// Mitsubishi GX Works2 project: Project34   PLC: FX3G

// global labels: Global1
VAR_GLOBAL
  StartA AT X010 : BOOL;
  SEN_IN AT X001 : BOOL;
  SEN_OUT AT X004 : BOOL;
  SEN_30 AT X003 : BOOL;
  SEN_15 AT X002 : BOOL;
  help1 AT M1 : BOOL;
END_VAR
VAR_GLOBAL CONSTANT
  Time1 : INT := 10;
  Time2 : INT := 10;
END_VAR
VAR_GLOBAL
  yuval AT X006 : BOOL;
END_VAR
VAR_GLOBAL CONSTANT
  Time3 : INT := 40;
END_VAR
VAR_GLOBAL
  ZILUF2 AT TS3 : BOOL;
  HELP3 AT M2 : BOOL;
  StartCoating AT X006 : BOOL;
  analogInput1 AT D8280 : INT;
  saveAnalogInput1 AT D8201 : INT;
END_VAR
VAR_GLOBAL CONSTANT
  topBound1 : INT := 5;
  topBound2 : INT := 10;
  lowerBound2 : INT := 6;
  Time4 : INT := 50;
END_VAR
VAR_GLOBAL
  CoatingLamp AT Y003 : BOOL;
  kkk1 AT Y002 : BOOL;
  kkk7 AT Y002 : BOOL;
  GFDKDN AT Y005 : BOOL;
  StartPacking AT X000 : BOOL;
  CreamStock AT D1100 : INT;
  UpdateCream AT D1200 : INT;
END_VAR
VAR_GLOBAL CONSTANT
  MinCream : INT := 300;
END_VAR
VAR_GLOBAL
  ChocolateStock AT D2100 : INT;
END_VAR
VAR_GLOBAL CONSTANT
  MinChocolate : INT := 240;
END_VAR
VAR_GLOBAL
  BiscuitStock AT D3100 : INT;
  UpdateBiscuit AT D3200 : INT;
END_VAR
VAR_GLOBAL CONSTANT
  MinBiscuit : INT := 6;
END_VAR
VAR_GLOBAL
  StartProcess AT X007 : BOOL;
  Check AT Y007 : BOOL;
  Coil5 AT M5 : BOOL;
  TransferCream AT X011 : BOOL;
  SprinklingContainer AT D4100 : INT;
  UpdateSprinkling AT D4200 : INT;
  ImmersionContainer AT D5100 : INT;
END_VAR
VAR_GLOBAL CONSTANT
  CreamUsed : INT := 300;
  NormalCoating : INT := 120;
  DoubleCoating : INT := 240;
  Init : INT;
  Unit : INT := 400;
END_VAR
VAR_GLOBAL
  Input AT D6000 : INT;
  UpdateChocolate AT D2300 : INT;
  UpdateImmersion AT D5300 : INT;
  BDIKA AT M8 : BOOL;
  DANUS AT M9 : BOOL;
  pack AT X000 : BOOL;
  Counter1 AT CC1 : BOOL;
END_VAR
VAR_GLOBAL CONSTANT
  counterVal1 : INT := 5;
END_VAR
VAR_GLOBAL
  Counter2 AT CC2 : BOOL;
END_VAR
VAR_GLOBAL CONSTANT
  counterVal2 : INT := 6;
END_VAR
VAR_GLOBAL
  Counter2output AT CS2 : BOOL;
  packCoil AT Y002 : BOOL;
  Krembows AT D3333 : INT;
END_VAR
VAR_GLOBAL CONSTANT
  addKrembow : INT := 6;
  Tens : INT := 10;
END_VAR
VAR_GLOBAL
  Coil12 AT M12 : BOOL;
  Coil13 AT M13 : BOOL;
END_VAR
VAR_GLOBAL CONSTANT
  Time5 : INT := 30;
END_VAR
VAR_GLOBAL
  Timer5 AT TC5 : BOOL;
  Coil14 AT M14 : BOOL;
  Coil15 AT M15 : BOOL;
  Timer6 AT TC6 : BOOL;
END_VAR
VAR_GLOBAL CONSTANT
  Time6 : INT := 10;
END_VAR
VAR_GLOBAL
  Timer7 AT TC7 : BOOL;
  Timer7Output AT TS7 : BOOL;
  Coil16 AT M16 : BOOL;
  Coil17 AT M17 : BOOL;
  Coil18 AT M18 : BOOL;
  Coil19 AT M19 : BOOL;
  Coil20 AT M20 : BOOL;
  Coil21 AT M21 : BOOL;
  Coil22 AT M22 : BOOL;
END_VAR
VAR_GLOBAL CONSTANT
  BiscuitUsed : INT := 6;
END_VAR
VAR_GLOBAL
  AnalogOutput AT D8282 : INT;
  Counter_Update AT CC8 : BOOL;
  Counter_Update6 AT CC9 : BOOL;
  Coil23 AT M23 : BOOL;
  Coil24 AT M24 : BOOL;
  Coil25 AT M25 : BOOL;
  Coil26 AT M26 : BOOL;
  WorkingDay AT Y007 : BOOL;
  Timer5Output AT TS5 : BOOL;
  Timer6Output AT TS6 : BOOL;
  DozensKrembows AT D4444 : INT;
  SprinklerFault AT X005 : BOOL;
  SprinklingLamp AT Y004 : BOOL;
  Timer3 AT TC3 : BOOL;
  Timer3Output AT TS3 : BOOL;
  Timer1 AT TC1 : BOOL;
  Timer1Output AT TS1 : BOOL;
  Timer2 AT TC2 : BOOL;
  Timer2Output AT TS2 : BOOL;
  ShinuaLamp1 AT Y000 : BOOL;
  ShinuaLamp2 AT Y001 : BOOL;
  Coil10 AT M10 : BOOL;
  Coil11 AT M11 : BOOL;
  Timer4 AT TC4 : BOOL;
  Timer4Output AT TS4 : BOOL;
  Counter1output AT CS1 : BOOL;
  Coil0 AT M0 : BOOL;
  coil27 AT M27 : BOOL;
END_VAR
VAR_GLOBAL CONSTANT
  Multiplier : INT := 40;
END_VAR
VAR_GLOBAL
  Coil28 AT M28 : BOOL;
END_VAR

// task Task_01 (event TRUE, interval 0, priority 31): POU_01

PROGRAM POU_01
(* structured ladder/FBD written out as ST: instructions are called as NAME(EN, inputs, outputs); _pN, _eN, _tN stand for wires *)
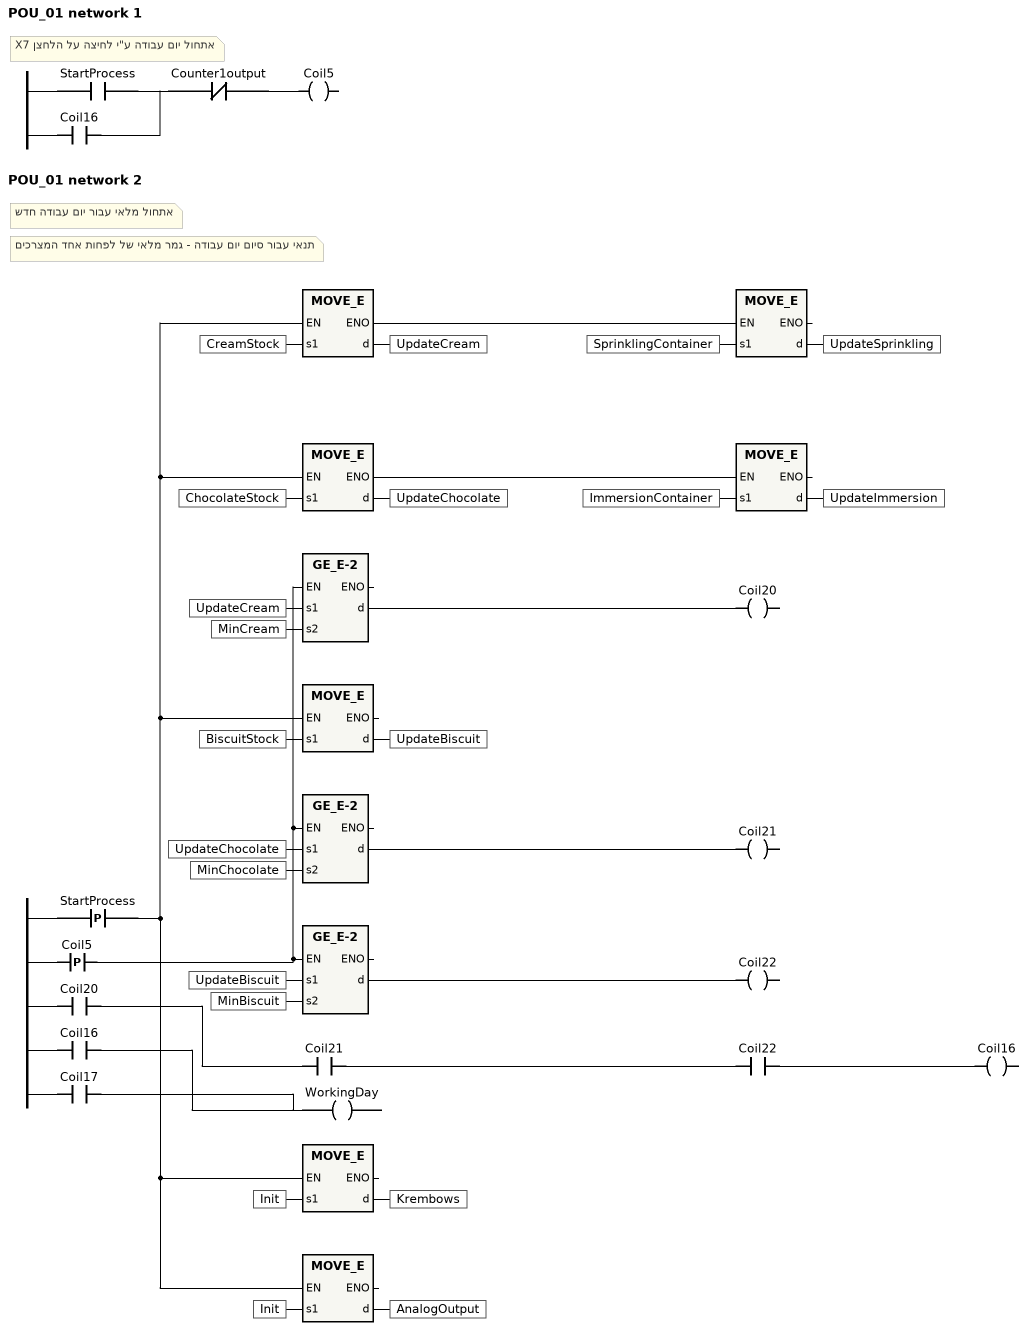
(* network 1 *)
(* אתחול יום עבודה ע"י לחיצה על הלחצן X7 *)
Coil5 := (StartProcess OR Coil16) AND NOT Counter1output;
(* network 2 *)
(* אתחול מלאי עבור יום עבודה חדש *)
(* תנאי עבור סיום יום עבודה - גמר מלאי של לפחות אחד המצרכים *)
_p1 := LDP(TRUE, StartProcess);
_e2 := MOVE_E(_p1, CreamStock, UpdateCream);
MOVE_E(_e2, SprinklingContainer, UpdateSprinkling);
_e3 := MOVE_E(_p1, ChocolateStock, UpdateChocolate);
MOVE_E(_e3, ImmersionContainer, UpdateImmersion);
MOVE_E(_p1, BiscuitStock, UpdateBiscuit);
MOVE_E(_p1, Init, Krembows);
MOVE_E(_p1, Init, AnalogOutput);
_p4 := LDP(TRUE, Coil5);
GE_E(_p4, UpdateCream, MinCream, _t5);
Coil20 := _t5;
GE_E(_p4, UpdateChocolate, MinChocolate, _t6);
Coil21 := _t6;
GE_E(_p4, UpdateBiscuit, MinBiscuit, _t7);
Coil22 := _t7;
Coil16 := Coil20 AND Coil21 AND Coil22;
WorkingDay := Coil16 OR Coil17;
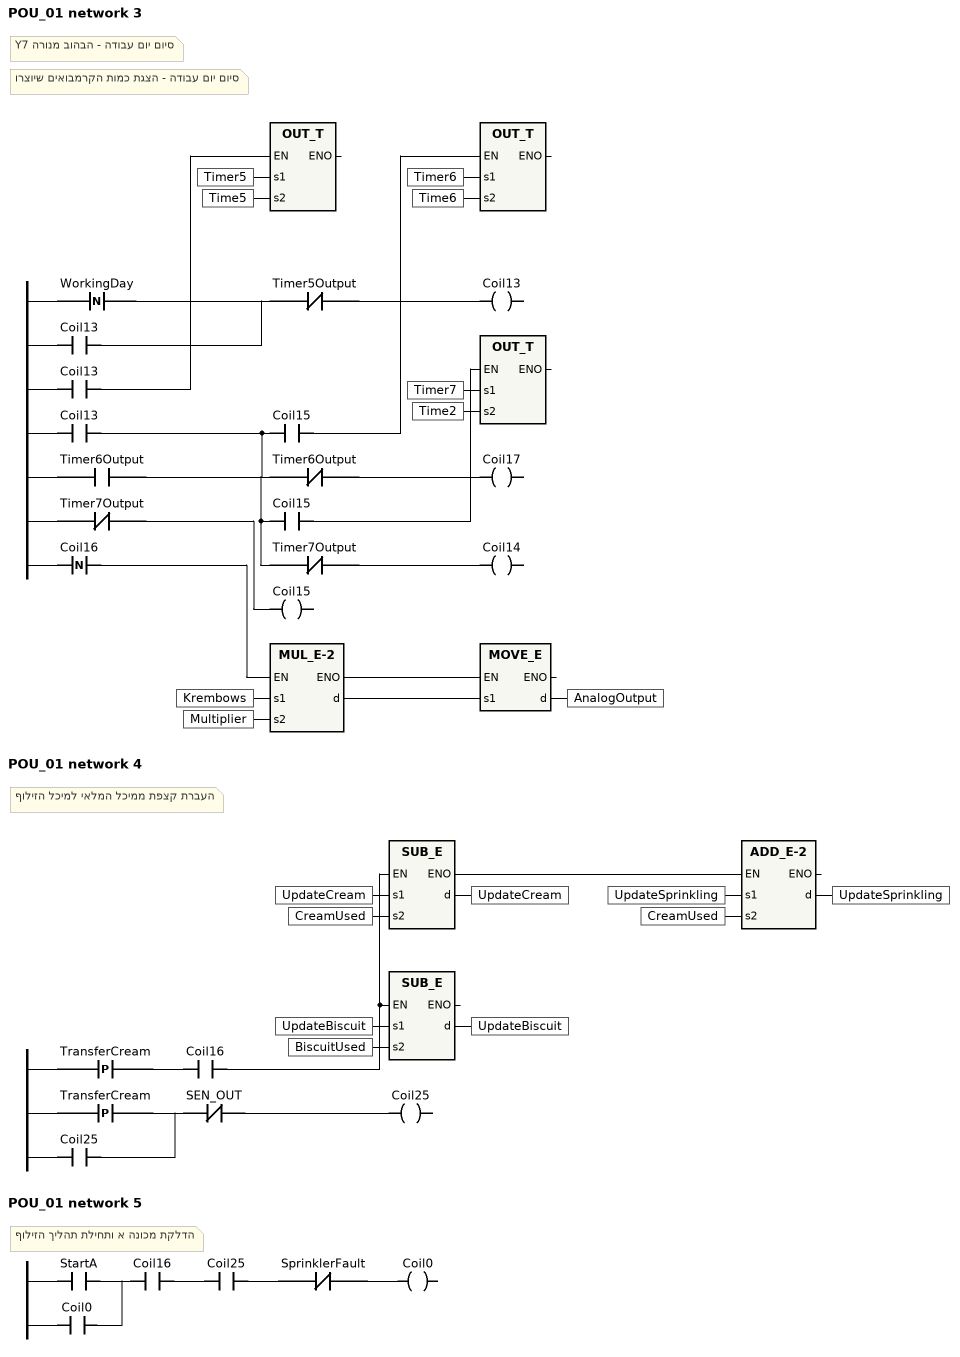
(* network 3 *)
(* סיום יום עבודה - הבהוב מנורה Y7 *)
(* סיום יום עבודה - הצגת כמות הקרמבואים שיוצרו *)
Coil13 := (LDF(TRUE, WorkingDay) OR Coil13) AND NOT Timer5Output;
OUT_T(Coil13, Timer5, Time5);
OUT_T(Coil13 AND Coil15, Timer6, Time6);
Coil17 := Coil13 AND NOT Timer6Output;
OUT_T(Timer6Output AND Coil15, Timer7, Time2);
Coil14 := Timer6Output AND NOT Timer7Output;
Coil15 := NOT Timer7Output;
_e2 := MUL_E(LDF(TRUE, Coil16), Krembows, Multiplier, _t1);
MOVE_E(_e2, _t1, AnalogOutput);
(* network 4 *)
(* העברת קצפת ממיכל המלאי למיכל הזילוף *)
_p1 := LDP(TRUE, TransferCream) AND Coil16;
_e2 := SUB_E(_p1, UpdateCream, CreamUsed, UpdateCream);
ADD_E(_e2, UpdateSprinkling, CreamUsed, UpdateSprinkling);
SUB_E(_p1, UpdateBiscuit, BiscuitUsed, UpdateBiscuit);
Coil25 := (LDP(TRUE, TransferCream) OR Coil25) AND NOT SEN_OUT;
(* network 5 *)
(* הדלקת מכונה א ותחילת תהליך הזילוף *)
Coil0 := (((StartA OR Coil0) AND Coil16) AND Coil25) AND NOT SprinklerFault;
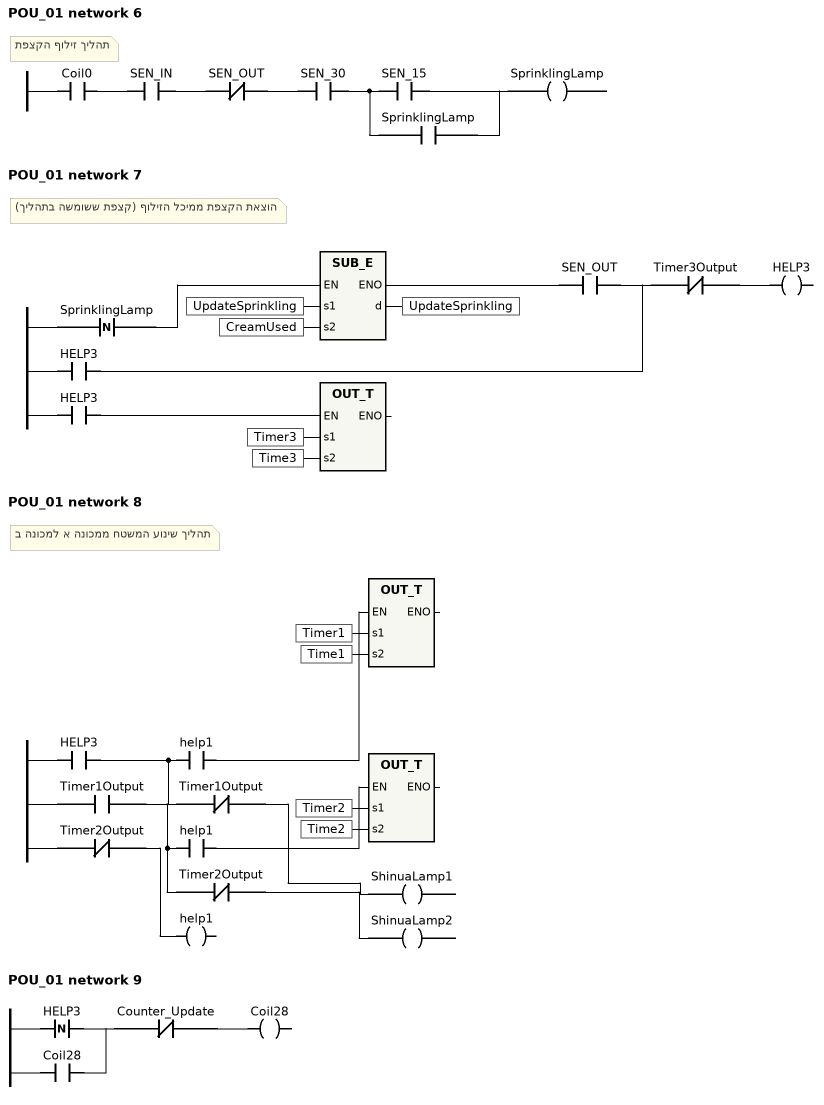
(* network 6 *)
(* תהליך זילוף הקצפת *)
_p1 := Coil0 AND SEN_IN AND NOT SEN_OUT AND SEN_30;
SprinklingLamp := (_p1 AND SEN_15) OR (_p1 AND SprinklingLamp);
(* network 7 *)
(* הוצאת הקצפת ממיכל הזילוף (קצפת ששומשה בתהליך) *)
_e1 := SUB_E(LDF(TRUE, SprinklingLamp), UpdateSprinkling, CreamUsed, UpdateSprinkling);
HELP3 := ((_e1 AND SEN_OUT) OR HELP3) AND NOT Timer3Output;
OUT_T(HELP3, Timer3, Time3);
(* network 8 *)
(* תהליך שינוע המשטח ממכונה א למכונה ב *)
OUT_T(HELP3 AND help1, Timer1, Time1);
ShinuaLamp1 := HELP3 AND NOT Timer1Output;
OUT_T(Timer1Output AND help1, Timer2, Time2);
ShinuaLamp2 := Timer1Output AND NOT Timer2Output;
help1 := NOT Timer2Output;
(* network 9 *)
Coil28 := (LDF(TRUE, HELP3) OR Coil28) AND NOT Counter_Update;
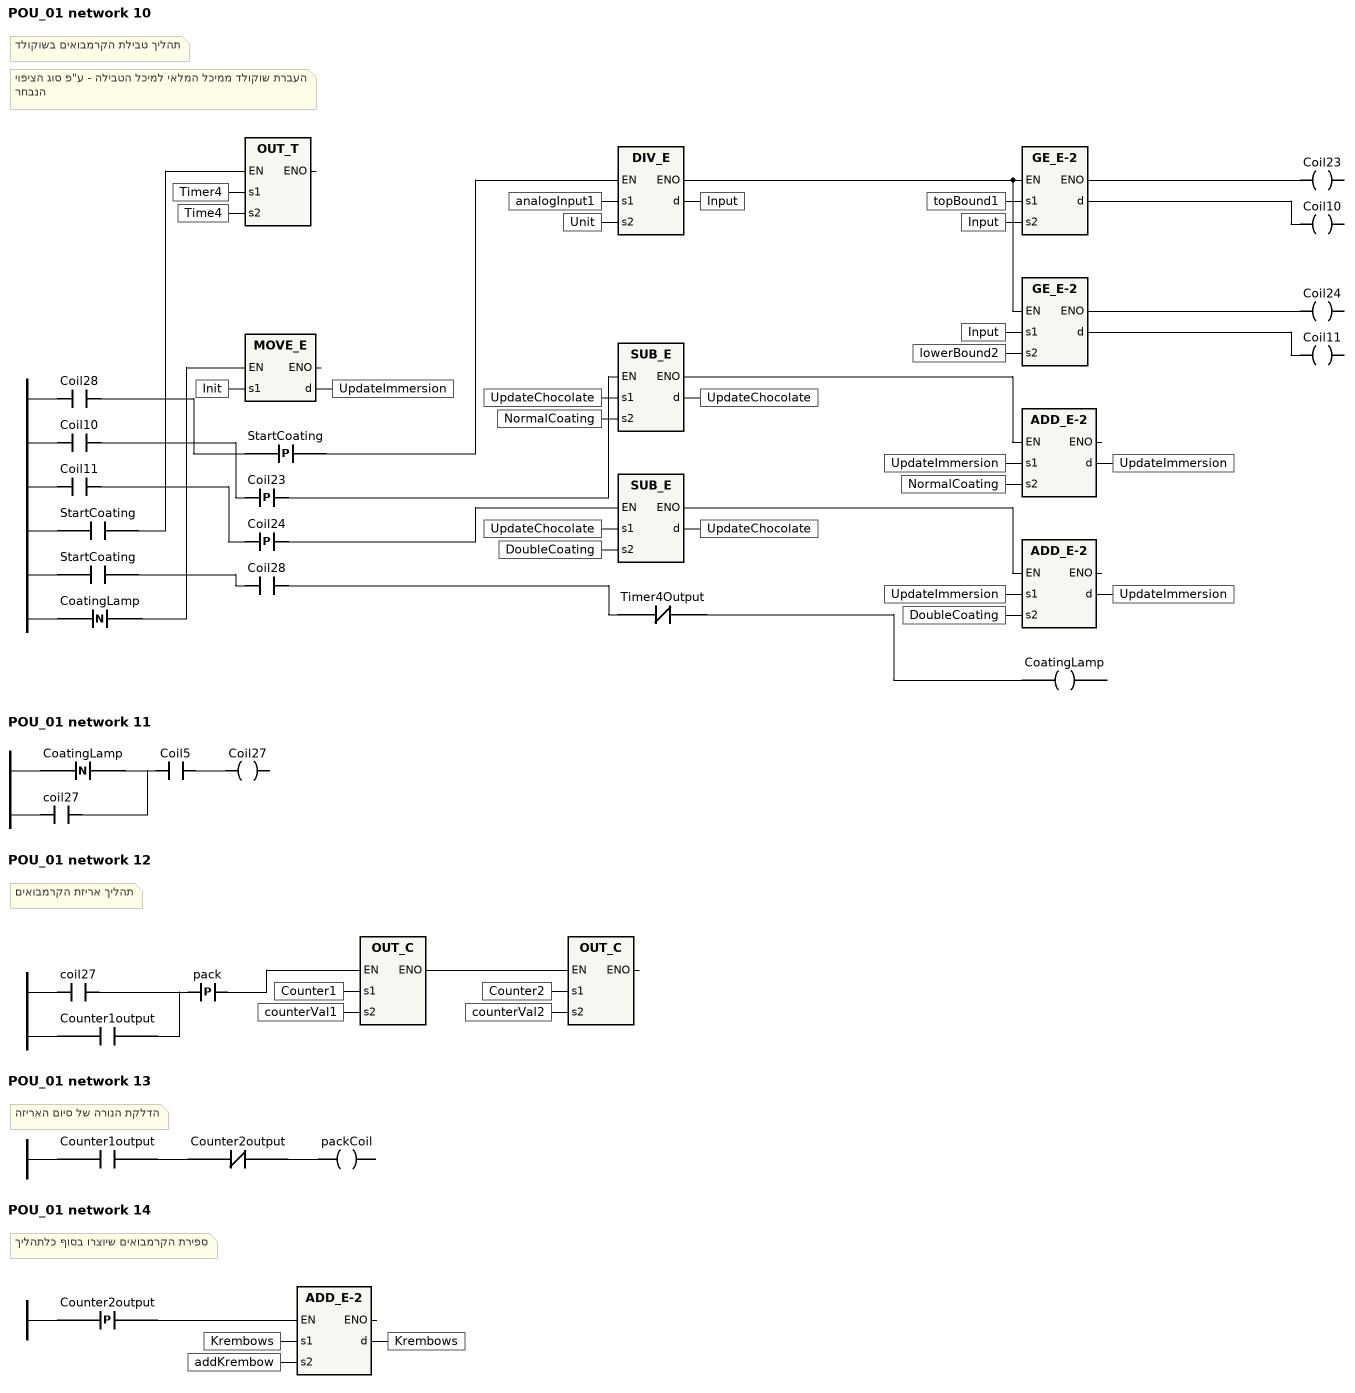
(* network 10 *)
(* תהליך טבילת הקרמבואים בשוקולד *)
(* העברת שוקולד ממיכל המלאי למיכל הטבילה - ע"פ סוג הציפוי הנבחר *)
_e1 := DIV_E(Coil28 AND LDP(TRUE, StartCoating), analogInput1, Unit, Input);
_e3 := GE_E(_e1, topBound1, Input, _t2);
Coil23 := _e3;
Coil10 := _t2;
_e5 := GE_E(_e1, Input, lowerBound2, _t4);
Coil24 := _e5;
Coil11 := _t4;
_e6 := SUB_E(Coil10 AND LDP(TRUE, Coil23), UpdateChocolate, NormalCoating, UpdateChocolate);
ADD_E(_e6, UpdateImmersion, NormalCoating, UpdateImmersion);
_e7 := SUB_E(Coil11 AND LDP(TRUE, Coil24), UpdateChocolate, DoubleCoating, UpdateChocolate);
ADD_E(_e7, UpdateImmersion, DoubleCoating, UpdateImmersion);
OUT_T(StartCoating, Timer4, Time4);
CoatingLamp := StartCoating AND Coil28 AND NOT Timer4Output;
MOVE_E(LDF(TRUE, CoatingLamp), Init, UpdateImmersion);
(* network 11 *)
Coil27 := (LDF(TRUE, CoatingLamp) OR coil27) AND Coil5;
(* network 12 *)
(* תהליך אריזת הקרמבואים *)
_e1 := OUT_C((coil27 OR Counter1output) AND LDP(TRUE, pack), Counter1, counterVal1);
OUT_C(_e1, Counter2, counterVal2);
(* network 13 *)
(* הדלקת הנורה של סיום האריזה *)
packCoil := Counter1output AND NOT Counter2output;
(* network 14 *)
(* ספירת הקרמבואים שיוצרו בסוף כלתהליך *)
ADD_E(LDP(TRUE, Counter2output), Krembows, addKrembow, Krembows);
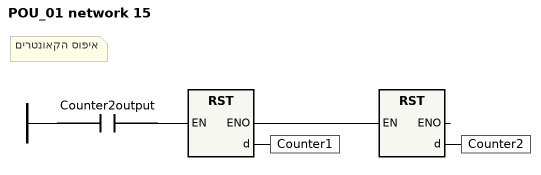
(* network 15 *)
(* איפוס הקאונטרים *)
_e1 := RST(Counter2output, Counter1);
RST(_e1, Counter2);
END_PROGRAM
